# EPICS substitutions: hugo/source/db/Beckhoff_6XXX/ecmcEL6002.substitutions
file "ecmcEL60X2-chX.template"
{
  pattern {CH_ID, NELM }
          {01,     22   }
          {02,     22   }
}
